# EPICS StreamDevice protocol: powerPMACApp/protocols/ppmac.proto
# PowerPMAC generic protocol file

InTerminator = CR LF;
OutTerminator = CR;
ExtraInput = Ignore;

getIntVar
{
  out "\$1";
  in "\n\$1=%d";
}

setIntVar
{
  out "\$1=%d";
  in "\n";
  @init { getIntVar; }
}

getFloatVar
{
  out "\$1";
  in "\n\$1=%f";
}

setFloatVar
{
  out "\$1=%f";
  in "\n";
  @init { getFloatVar; }
}
